# EPICS autosave request: iocBoot/sioc-esb-hvfb01/hvfb.req
$(P):UPDATE_TIME
$(P):INT_TIME
$(P):VDES
$(P):VMAX
$(P):SMOOTHING
$(P):CFACT
$(P):OUT_NOM
